// TIA Portal V18 export
DATA_BLOCK "AXIS_Z1_V2_CMMS"   // DB66
VERSION : 0.1
// stored: AutoNumber true, DBAccessibleFromOPCUA true, InstanceOfName AXIS_CMMT_V2_Motion_Control, InstanceOfType FB
"AXIS_CMMT_V2_Motion_Control"
   // VAR_INPUT
   //    DriverType : String;
   //    EnableAxis : Bool;
   //    PrintingModeWebDB : Int;
   //    PositionWebDB : DInt;
   //    VelocityWebDB : Real;
   //    Stop : Bool;
   //    EmergencyStop : Bool;
   //    JogPos : Bool;
   //    JogNeg : Bool;
   //    AckError : Bool;
   //    ConfigEPos : DWord;
   //    PosMin : DInt;
   //    PosMax : DInt;
   //    Jogging : Bool;
   //    MarginSoft : DInt;
   //    MarginHard : DInt;
   //    MotionLock : Bool;
   //    AXISEnabled : Bool;
   //    AXISPosOk : Bool;
   //    AXISReference : Bool;
   //    AXISAxisWarning : Bool;
   //    AXISAxisError : Bool;
   //    AXISLockout : Bool;
   //    AXISActVelocity : Real;
   //    AXISActPosition : DInt;
   //    AXISAxisAckSetpoint : Bool;
   //    AXISReady4Motion : Bool;
   //    AXISEposZSW1 : Word;
   //    AXISStatus : Word;
   //    JogStartPos : DInt;
   //    JogEndPos : DInt;
   //    AxisType : Int;
   //    YPosition : DInt;
   //    PositionDelay : Bool;
   //    NoGoZoneActive : Bool;
   //    NoGoZoneHomingPermission : Bool;
   //    NoGoZoneMovePermission : Bool;
   //    NoGoZoneJogPosPermission : Bool;
   //    NoGoZoneJogNegPermission : Bool;
   //    RMPositioningError : DInt;
   //    MachineStart : Bool;
   // END_VAR
   // VAR_OUTPUT
   //    Status : Word;
   //    Overrange : Bool;
   //    Ready : Bool;
   //    DriveMoving : Bool;
   //    DriveStop : Bool;
   //    Standstill : Bool;
   //    MC : Bool;
   //    AXISModePos : Int;
   //    AXISEnableAxis : Bool;
   //    AXISCancelTraversing : Bool;
   //    AXISIntermediateStop : Bool;
   //    AXISJog1 : Bool;
   //    AXISJog2 : Bool;
   //    AXISAckError : Bool;
   //    AXISExecuteMode : Bool;
   //    AXISPosition : DInt;
   //    AXISVelocity : Real;
   //    AXISConfigEpos : DWord;
   //    AXISRelative : Bool;
   //    AXISHoming : Bool;
   //    FinishTask_Delay : Bool;
   // END_VAR
   // VAR_IN_OUT
   //    StartTask : Bool;
   //    Execute : Bool;
   //    Homing : Bool;
   //    Printing : Bool;
   // END_VAR
   // VAR
   //    ExecutingMemory : Bool;
   //    HomingMemory : Bool;
   //    TaskMemory : Bool;
   //    ModePos : Int;
   //    PosOk : Bool;
   //    Reference : Bool;
   //    PositionInternal : DInt;
   //    LockoutInternal : Bool;
   //    RelativeMode : Bool;
   //    AbsoluteMode : Bool;
   //    TaskFinished : Bool;
   //    JoggingXPermission : Bool;
   //    JoggingYPermission : Bool;
   //    JoggingPOSZ1Z2Permission : Bool;
   //    JoggingNEGZ1Z2Permission : Bool;
   //    JoggingPosMax : DInt;
   //    JoggingPosMin : DInt;
   //    JoggingPositionCorrection : DInt;
   //    ProfinetDisconnected : Bool;
   //    PositionStepPlus : DInt;
   //    CMMT : Bool;
   //    CMMS : Bool;
   //    RMStepStartPosition : DInt;
   //    RMPredictedPosition : DInt;
   //    RMFinalPosition : DInt;
   //    RMLastStepPositionError : DInt;
   //    RMStartTaskM01 : Bool;
   //    RMStartTaksM02 : Bool;
   //    RMStepRangePlus : DInt;
   //    RMStepRangeMinus : DInt;
   //    RelativeDirectionInRange : Bool;
   // END_VAR
BEGIN
END_DATA_BLOCK
